TYPE StepperSTMControl :
STRUCT
	Enable : BOOL;
	Reset : BOOL;
	ReduceTorque : BOOL;
	DigitalOutput1 : BOOL;
END_STRUCT
END_TYPE

(* stored: Version 1.1.0.1, ProductVersion 3.1.4024.11
   DUT StepperSTMControl: Id {088d4595-d08e-4f88-af28-e4c50a5451e6} *)
